KUKA KRL program: sPlanen2.src, sPlanen2.dat

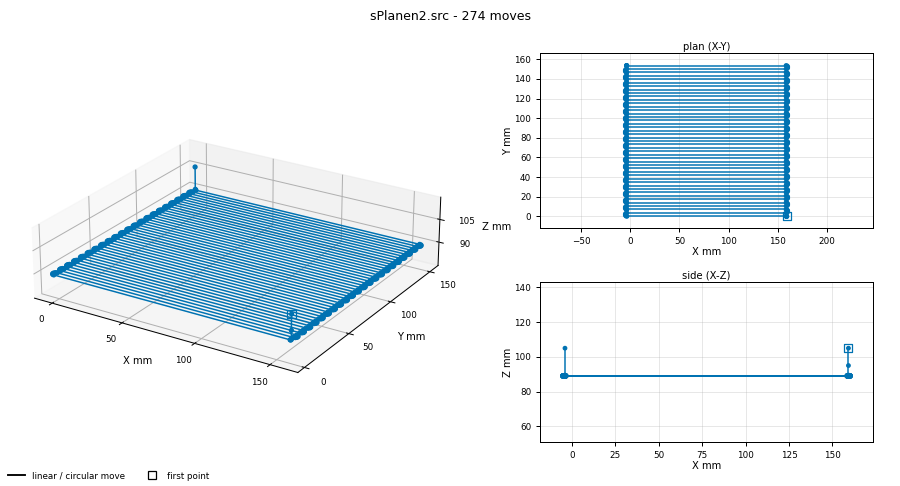
[picture p0: tool path of sPlanen2.src, 274 of 275 moves have a stored position in this frame; points joined in program order, loops and branches not executed]
--- sPlanen2.src ---
&ACCESS RVO
DEF sPlanen2()
; Generated by AUTODESK Fusion 360 CAM 2.0.14793
; Creation date: Thursday, March 16, 2023 18:51:23
;FOLD sPlanen2
; Start position (joint) = {A1 5,A2 -80,A3 100,A4 75,A5 -60,A6 -65}
; Tool Number            = 4
; Base Number            = 1
; Spindle Speed          = 5000 RPM
; Program file name      = sPlanen2.src

PTP {A1 5,A2 -80,A3 100,A4 75,A5 -60,A6 -65,E1 0,E2 0,E3 0,E4 0,E5 0,E6 0}
$VEL.CP=0.02
LIN {X 159.250,Y 0.025,Z 105.000,A 180.000,B 0.000,C 180.000} C_DIS
LIN {X 159.250,Y 0.025,Z 95.000,A 180.000,B 0.000,C 180.000} C_DIS
; Plunge Move Starts
$VEL.CP=0.01
LIN {X 159.250,Y 0.025,Z 89.500,A 180.000,B 0.000,C 180.000} C_DIS
; Lead In Move Starts
LIN {X 159.104,Y 0.025,Z 89.146,A 180.000,B 0.000,C 180.000} C_DIS
LIN {X 158.750,Y 0.025,Z 89.000,A 180.000,B 0.000,C 180.000} C_DIS
LIN {X 158.510,Y 0.025,Z 89.000,A 180.000,B 0.000,C 180.000} C_DIS
; Cutting Move Starts
$VEL.CP=0.02
LIN {X -3.510,Y 0.025,Z 89.000,A 180.000,B 0.000,C 180.000} C_DIS
; Link Move Starts
LIN {X -4.536,Y 0.358,Z 89.000,A 180.000,B 0.000,C 180.000} C_DIS
LIN {X -5.170,Y 1.231,Z 89.000,A 180.000,B 0.000,C 180.000} C_DIS
LIN {X -5.170,Y 2.309,Z 89.000,A 180.000,B 0.000,C 180.000} C_DIS
LIN {X -4.536,Y 3.182,Z 89.000,A 180.000,B 0.000,C 180.000} C_DIS
LIN {X -3.510,Y 3.515,Z 89.000,A 180.000,B 0.000,C 180.000} C_DIS
; Cutting Move Starts
LIN {X 158.510,Y 3.515,Z 89.000,A 180.000,B 0.000,C 180.000} C_DIS
; Link Move Starts
LIN {X 159.536,Y 3.848,Z 89.000,A 180.000,B 0.000,C 180.000} C_DIS
LIN {X 160.170,Y 4.721,Z 89.000,A 180.000,B 0.000,C 180.000} C_DIS
LIN {X 160.170,Y 5.800,Z 89.000,A 180.000,B 0.000,C 180.000} C_DIS
LIN {X 159.536,Y 6.672,Z 89.000,A 180.000,B 0.000,C 180.000} C_DIS
LIN {X 158.510,Y 7.005,Z 89.000,A 180.000,B 0.000,C 180.000} C_DIS
; Cutting Move Starts
LIN {X -3.510,Y 7.005,Z 89.000,A 180.000,B 0.000,C 180.000} C_DIS
; Link Move Starts
LIN {X -4.536,Y 7.339,Z 89.000,A 180.000,B 0.000,C 180.000} C_DIS
LIN {X -5.170,Y 8.211,Z 89.000,A 180.000,B 0.000,C 180.000} C_DIS
LIN {X -5.170,Y 9.290,Z 89.000,A 180.000,B 0.000,C 180.000} C_DIS
LIN {X -4.536,Y 10.162,Z 89.000,A 180.000,B 0.000,C 180.000} C_DIS
LIN {X -3.510,Y 10.495,Z 89.000,A 180.000,B 0.000,C 180.000} C_DIS
; Cutting Move Starts
LIN {X 158.510,Y 10.495,Z 89.000,A 180.000,B 0.000,C 180.000} C_DIS
; Link Move Starts
LIN {X 159.536,Y 10.829,Z 89.000,A 180.000,B 0.000,C 180.000} C_DIS
LIN {X 160.170,Y 11.701,Z 89.000,A 180.000,B 0.000,C 180.000} C_DIS
LIN {X 160.170,Y 12.780,Z 89.000,A 180.000,B 0.000,C 180.000} C_DIS
LIN {X 159.536,Y 13.652,Z 89.000,A 180.000,B 0.000,C 180.000} C_DIS
LIN {X 158.510,Y 13.986,Z 89.000,A 180.000,B 0.000,C 180.000} C_DIS
; Cutting Move Starts
LIN {X -3.510,Y 13.986,Z 89.000,A 180.000,B 0.000,C 180.000} C_DIS
; Link Move Starts
LIN {X -4.536,Y 14.319,Z 89.000,A 180.000,B 0.000,C 180.000} C_DIS
LIN {X -5.170,Y 15.191,Z 89.000,A 180.000,B 0.000,C 180.000} C_DIS
LIN {X -5.170,Y 16.270,Z 89.000,A 180.000,B 0.000,C 180.000} C_DIS
LIN {X -4.536,Y 17.142,Z 89.000,A 180.000,B 0.000,C 180.000} C_DIS
LIN {X -3.510,Y 17.476,Z 89.000,A 180.000,B 0.000,C 180.000} C_DIS
; Cutting Move Starts
LIN {X 158.510,Y 17.476,Z 89.000,A 180.000,B 0.000,C 180.000} C_DIS
; Link Move Starts
LIN {X 159.536,Y 17.809,Z 89.000,A 180.000,B 0.000,C 180.000} C_DIS
LIN {X 160.170,Y 18.681,Z 89.000,A 180.000,B 0.000,C 180.000} C_DIS
LIN {X 160.170,Y 19.760,Z 89.000,A 180.000,B 0.000,C 180.000} C_DIS
LIN {X 159.536,Y 20.633,Z 89.000,A 180.000,B 0.000,C 180.000} C_DIS
LIN {X 158.510,Y 20.966,Z 89.000,A 180.000,B 0.000,C 180.000} C_DIS
; Cutting Move Starts
LIN {X -3.510,Y 20.966,Z 89.000,A 180.000,B 0.000,C 180.000} C_DIS
; Link Move Starts
LIN {X -4.536,Y 21.299,Z 89.000,A 180.000,B 0.000,C 180.000} C_DIS
LIN {X -5.170,Y 22.172,Z 89.000,A 180.000,B 0.000,C 180.000} C_DIS
LIN {X -5.170,Y 23.250,Z 89.000,A 180.000,B 0.000,C 180.000} C_DIS
LIN {X -4.536,Y 24.123,Z 89.000,A 180.000,B 0.000,C 180.000} C_DIS
LIN {X -3.510,Y 24.456,Z 89.000,A 180.000,B 0.000,C 180.000} C_DIS
; Cutting Move Starts
LIN {X 158.510,Y 24.456,Z 89.000,A 180.000,B 0.000,C 180.000} C_DIS
; Link Move Starts
LIN {X 159.536,Y 24.789,Z 89.000,A 180.000,B 0.000,C 180.000} C_DIS
LIN {X 160.170,Y 25.662,Z 89.000,A 180.000,B 0.000,C 180.000} C_DIS
LIN {X 160.170,Y 26.740,Z 89.000,A 180.000,B 0.000,C 180.000} C_DIS
LIN {X 159.536,Y 27.613,Z 89.000,A 180.000,B 0.000,C 180.000} C_DIS
LIN {X 158.510,Y 27.946,Z 89.000,A 180.000,B 0.000,C 180.000} C_DIS
; Cutting Move Starts
LIN {X -3.510,Y 27.946,Z 89.000,A 180.000,B 0.000,C 180.000} C_DIS
; Link Move Starts
LIN {X -4.536,Y 28.279,Z 89.000,A 180.000,B 0.000,C 180.000} C_DIS
LIN {X -5.170,Y 29.152,Z 89.000,A 180.000,B 0.000,C 180.000} C_DIS
LIN {X -5.170,Y 30.230,Z 89.000,A 180.000,B 0.000,C 180.000} C_DIS
LIN {X -4.536,Y 31.103,Z 89.000,A 180.000,B 0.000,C 180.000} C_DIS
LIN {X -3.510,Y 31.436,Z 89.000,A 180.000,B 0.000,C 180.000} C_DIS
; Cutting Move Starts
LIN {X 158.510,Y 31.436,Z 89.000,A 180.000,B 0.000,C 180.000} C_DIS
; Link Move Starts
LIN {X 159.536,Y 31.769,Z 89.000,A 180.000,B 0.000,C 180.000} C_DIS
LIN {X 160.170,Y 32.642,Z 89.000,A 180.000,B 0.000,C 180.000} C_DIS
LIN {X 160.170,Y 33.720,Z 89.000,A 180.000,B 0.000,C 180.000} C_DIS
LIN {X 159.536,Y 34.593,Z 89.000,A 180.000,B 0.000,C 180.000} C_DIS
LIN {X 158.510,Y 34.926,Z 89.000,A 180.000,B 0.000,C 180.000} C_DIS
; Cutting Move Starts
LIN {X -3.510,Y 34.926,Z 89.000,A 180.000,B 0.000,C 180.000} C_DIS
; Link Move Starts
LIN {X -4.536,Y 35.259,Z 89.000,A 180.000,B 0.000,C 180.000} C_DIS
LIN {X -5.170,Y 36.132,Z 89.000,A 180.000,B 0.000,C 180.000} C_DIS
LIN {X -5.170,Y 37.211,Z 89.000,A 180.000,B 0.000,C 180.000} C_DIS
LIN {X -4.536,Y 38.083,Z 89.000,A 180.000,B 0.000,C 180.000} C_DIS
LIN {X -3.510,Y 38.416,Z 89.000,A 180.000,B 0.000,C 180.000} C_DIS
; Cutting Move Starts
LIN {X 158.510,Y 38.416,Z 89.000,A 180.000,B 0.000,C 180.000} C_DIS
; Link Move Starts
LIN {X 159.536,Y 38.750,Z 89.000,A 180.000,B 0.000,C 180.000} C_DIS
LIN {X 160.170,Y 39.622,Z 89.000,A 180.000,B 0.000,C 180.000} C_DIS
LIN {X 160.170,Y 40.701,Z 89.000,A 180.000,B 0.000,C 180.000} C_DIS
LIN {X 159.536,Y 41.573,Z 89.000,A 180.000,B 0.000,C 180.000} C_DIS
LIN {X 158.510,Y 41.906,Z 89.000,A 180.000,B 0.000,C 180.000} C_DIS
; Cutting Move Starts
LIN {X -3.510,Y 41.906,Z 89.000,A 180.000,B 0.000,C 180.000} C_DIS
; Link Move Starts
LIN {X -4.536,Y 42.240,Z 89.000,A 180.000,B 0.000,C 180.000} C_DIS
LIN {X -5.170,Y 43.112,Z 89.000,A 180.000,B 0.000,C 180.000} C_DIS
LIN {X -5.170,Y 44.191,Z 89.000,A 180.000,B 0.000,C 180.000} C_DIS
LIN {X -4.536,Y 45.063,Z 89.000,A 180.000,B 0.000,C 180.000} C_DIS
LIN {X -3.510,Y 45.397,Z 89.000,A 180.000,B 0.000,C 180.000} C_DIS
; Cutting Move Starts
LIN {X 158.510,Y 45.397,Z 89.000,A 180.000,B 0.000,C 180.000} C_DIS
; Link Move Starts
LIN {X 159.536,Y 45.730,Z 89.000,A 180.000,B 0.000,C 180.000} C_DIS
LIN {X 160.170,Y 46.602,Z 89.000,A 180.000,B 0.000,C 180.000} C_DIS
LIN {X 160.170,Y 47.681,Z 89.000,A 180.000,B 0.000,C 180.000} C_DIS
LIN {X 159.536,Y 48.553,Z 89.000,A 180.000,B 0.000,C 180.000} C_DIS
LIN {X 158.510,Y 48.887,Z 89.000,A 180.000,B 0.000,C 180.000} C_DIS
; Cutting Move Starts
LIN {X -3.510,Y 48.887,Z 89.000,A 180.000,B 0.000,C 180.000} C_DIS
; Link Move Starts
LIN {X -4.536,Y 49.220,Z 89.000,A 180.000,B 0.000,C 180.000} C_DIS
LIN {X -5.170,Y 50.092,Z 89.000,A 180.000,B 0.000,C 180.000} C_DIS
LIN {X -5.170,Y 51.171,Z 89.000,A 180.000,B 0.000,C 180.000} C_DIS
LIN {X -4.536,Y 52.044,Z 89.000,A 180.000,B 0.000,C 180.000} C_DIS
LIN {X -3.510,Y 52.377,Z 89.000,A 180.000,B 0.000,C 180.000} C_DIS
; Cutting Move Starts
LIN {X 158.510,Y 52.377,Z 89.000,A 180.000,B 0.000,C 180.000} C_DIS
; Link Move Starts
LIN {X 159.536,Y 52.710,Z 89.000,A 180.000,B 0.000,C 180.000} C_DIS
LIN {X 160.170,Y 53.583,Z 89.000,A 180.000,B 0.000,C 180.000} C_DIS
LIN {X 160.170,Y 54.661,Z 89.000,A 180.000,B 0.000,C 180.000} C_DIS
LIN {X 159.536,Y 55.534,Z 89.000,A 180.000,B 0.000,C 180.000} C_DIS
LIN {X 158.510,Y 55.867,Z 89.000,A 180.000,B 0.000,C 180.000} C_DIS
; Cutting Move Starts
LIN {X -3.510,Y 55.867,Z 89.000,A 180.000,B 0.000,C 180.000} C_DIS
; Link Move Starts
LIN {X -4.536,Y 56.200,Z 89.000,A 180.000,B 0.000,C 180.000} C_DIS
LIN {X -5.170,Y 57.073,Z 89.000,A 180.000,B 0.000,C 180.000} C_DIS
LIN {X -5.170,Y 58.151,Z 89.000,A 180.000,B 0.000,C 180.000} C_DIS
LIN {X -4.536,Y 59.024,Z 89.000,A 180.000,B 0.000,C 180.000} C_DIS
LIN {X -3.510,Y 59.357,Z 89.000,A 180.000,B 0.000,C 180.000} C_DIS
; Cutting Move Starts
LIN {X 158.510,Y 59.357,Z 89.000,A 180.000,B 0.000,C 180.000} C_DIS
; Link Move Starts
LIN {X 159.536,Y 59.690,Z 89.000,A 180.000,B 0.000,C 180.000} C_DIS
LIN {X 160.170,Y 60.563,Z 89.000,A 180.000,B 0.000,C 180.000} C_DIS
LIN {X 160.170,Y 61.641,Z 89.000,A 180.000,B 0.000,C 180.000} C_DIS
LIN {X 159.536,Y 62.514,Z 89.000,A 180.000,B 0.000,C 180.000} C_DIS
LIN {X 158.510,Y 62.847,Z 89.000,A 180.000,B 0.000,C 180.000} C_DIS
; Cutting Move Starts
LIN {X -3.510,Y 62.847,Z 89.000,A 180.000,B 0.000,C 180.000} C_DIS
; Link Move Starts
LIN {X -4.536,Y 63.180,Z 89.000,A 180.000,B 0.000,C 180.000} C_DIS
LIN {X -5.170,Y 64.053,Z 89.000,A 180.000,B 0.000,C 180.000} C_DIS
LIN {X -5.170,Y 65.131,Z 89.000,A 180.000,B 0.000,C 180.000} C_DIS
LIN {X -4.536,Y 66.004,Z 89.000,A 180.000,B 0.000,C 180.000} C_DIS
LIN {X -3.510,Y 66.337,Z 89.000,A 180.000,B 0.000,C 180.000} C_DIS
; Cutting Move Starts
LIN {X 158.510,Y 66.337,Z 89.000,A 180.000,B 0.000,C 180.000} C_DIS
; Link Move Starts
LIN {X 159.536,Y 66.670,Z 89.000,A 180.000,B 0.000,C 180.000} C_DIS
LIN {X 160.170,Y 67.543,Z 89.000,A 180.000,B 0.000,C 180.000} C_DIS
LIN {X 160.170,Y 68.622,Z 89.000,A 180.000,B 0.000,C 180.000} C_DIS
LIN {X 159.536,Y 69.494,Z 89.000,A 180.000,B 0.000,C 180.000} C_DIS
LIN {X 158.510,Y 69.827,Z 89.000,A 180.000,B 0.000,C 180.000} C_DIS
; Cutting Move Starts
LIN {X -3.510,Y 69.827,Z 89.000,A 180.000,B 0.000,C 180.000} C_DIS
; Link Move Starts
LIN {X -4.536,Y 70.161,Z 89.000,A 180.000,B 0.000,C 180.000} C_DIS
LIN {X -5.170,Y 71.033,Z 89.000,A 180.000,B 0.000,C 180.000} C_DIS
LIN {X -5.170,Y 72.112,Z 89.000,A 180.000,B 0.000,C 180.000} C_DIS
LIN {X -4.536,Y 72.984,Z 89.000,A 180.000,B 0.000,C 180.000} C_DIS
LIN {X -3.510,Y 73.317,Z 89.000,A 180.000,B 0.000,C 180.000} C_DIS
; Cutting Move Starts
LIN {X 158.510,Y 73.317,Z 89.000,A 180.000,B 0.000,C 180.000} C_DIS
; Link Move Starts
LIN {X 159.536,Y 73.651,Z 89.000,A 180.000,B 0.000,C 180.000} C_DIS
LIN {X 160.170,Y 74.523,Z 89.000,A 180.000,B 0.000,C 180.000} C_DIS
LIN {X 160.170,Y 75.602,Z 89.000,A 180.000,B 0.000,C 180.000} C_DIS
LIN {X 159.536,Y 76.474,Z 89.000,A 180.000,B 0.000,C 180.000} C_DIS
LIN {X 158.510,Y 76.808,Z 89.000,A 180.000,B 0.000,C 180.000} C_DIS
; Cutting Move Starts
LIN {X -3.510,Y 76.808,Z 89.000,A 180.000,B 0.000,C 180.000} C_DIS
; Link Move Starts
LIN {X -4.536,Y 77.141,Z 89.000,A 180.000,B 0.000,C 180.000} C_DIS
LIN {X -5.170,Y 78.013,Z 89.000,A 180.000,B 0.000,C 180.000} C_DIS
LIN {X -5.170,Y 79.092,Z 89.000,A 180.000,B 0.000,C 180.000} C_DIS
LIN {X -4.536,Y 79.964,Z 89.000,A 180.000,B 0.000,C 180.000} C_DIS
LIN {X -3.510,Y 80.298,Z 89.000,A 180.000,B 0.000,C 180.000} C_DIS
; Cutting Move Starts
LIN {X 158.510,Y 80.298,Z 89.000,A 180.000,B 0.000,C 180.000} C_DIS
; Link Move Starts
LIN {X 159.536,Y 80.631,Z 89.000,A 180.000,B 0.000,C 180.000} C_DIS
LIN {X 160.170,Y 81.503,Z 89.000,A 180.000,B 0.000,C 180.000} C_DIS
LIN {X 160.170,Y 82.582,Z 89.000,A 180.000,B 0.000,C 180.000} C_DIS
LIN {X 159.536,Y 83.455,Z 89.000,A 180.000,B 0.000,C 180.000} C_DIS
LIN {X 158.510,Y 83.788,Z 89.000,A 180.000,B 0.000,C 180.000} C_DIS
; Cutting Move Starts
LIN {X -3.510,Y 83.788,Z 89.000,A 180.000,B 0.000,C 180.000} C_DIS
; Link Move Starts
LIN {X -4.536,Y 84.121,Z 89.000,A 180.000,B 0.000,C 180.000} C_DIS
LIN {X -5.170,Y 84.994,Z 89.000,A 180.000,B 0.000,C 180.000} C_DIS
LIN {X -5.170,Y 86.072,Z 89.000,A 180.000,B 0.000,C 180.000} C_DIS
LIN {X -4.536,Y 86.945,Z 89.000,A 180.000,B 0.000,C 180.000} C_DIS
LIN {X -3.510,Y 87.278,Z 89.000,A 180.000,B 0.000,C 180.000} C_DIS
; Cutting Move Starts
LIN {X 158.510,Y 87.278,Z 89.000,A 180.000,B 0.000,C 180.000} C_DIS
; Link Move Starts
LIN {X 159.536,Y 87.611,Z 89.000,A 180.000,B 0.000,C 180.000} C_DIS
LIN {X 160.170,Y 88.484,Z 89.000,A 180.000,B 0.000,C 180.000} C_DIS
LIN {X 160.170,Y 89.562,Z 89.000,A 180.000,B 0.000,C 180.000} C_DIS
LIN {X 159.536,Y 90.435,Z 89.000,A 180.000,B 0.000,C 180.000} C_DIS
LIN {X 158.510,Y 90.768,Z 89.000,A 180.000,B 0.000,C 180.000} C_DIS
; Cutting Move Starts
LIN {X -3.510,Y 90.768,Z 89.000,A 180.000,B 0.000,C 180.000} C_DIS
; Link Move Starts
LIN {X -4.536,Y 91.101,Z 89.000,A 180.000,B 0.000,C 180.000} C_DIS
LIN {X -5.170,Y 91.974,Z 89.000,A 180.000,B 0.000,C 180.000} C_DIS
LIN {X -5.170,Y 93.052,Z 89.000,A 180.000,B 0.000,C 180.000} C_DIS
LIN {X -4.536,Y 93.925,Z 89.000,A 180.000,B 0.000,C 180.000} C_DIS
LIN {X -3.510,Y 94.258,Z 89.000,A 180.000,B 0.000,C 180.000} C_DIS
; Cutting Move Starts
LIN {X 158.510,Y 94.258,Z 89.000,A 180.000,B 0.000,C 180.000} C_DIS
; Link Move Starts
LIN {X 159.536,Y 94.591,Z 89.000,A 180.000,B 0.000,C 180.000} C_DIS
LIN {X 160.170,Y 95.464,Z 89.000,A 180.000,B 0.000,C 180.000} C_DIS
LIN {X 160.170,Y 96.542,Z 89.000,A 180.000,B 0.000,C 180.000} C_DIS
LIN {X 159.536,Y 97.415,Z 89.000,A 180.000,B 0.000,C 180.000} C_DIS
LIN {X 158.510,Y 97.748,Z 89.000,A 180.000,B 0.000,C 180.000} C_DIS
; Cutting Move Starts
LIN {X -3.510,Y 97.748,Z 89.000,A 180.000,B 0.000,C 180.000} C_DIS
; Link Move Starts
LIN {X -4.536,Y 98.081,Z 89.000,A 180.000,B 0.000,C 180.000} C_DIS
LIN {X -5.170,Y 98.954,Z 89.000,A 180.000,B 0.000,C 180.000} C_DIS
LIN {X -5.170,Y 100.033,Z 89.000,A 180.000,B 0.000,C 180.000} C_DIS
LIN {X -4.536,Y 100.905,Z 89.000,A 180.000,B 0.000,C 180.000} C_DIS
LIN {X -3.510,Y 101.238,Z 89.000,A 180.000,B 0.000,C 180.000} C_DIS
; Cutting Move Starts
LIN {X 158.510,Y 101.238,Z 89.000,A 180.000,B 0.000,C 180.000} C_DIS
; Link Move Starts
LIN {X 159.536,Y 101.572,Z 89.000,A 180.000,B 0.000,C 180.000} C_DIS
LIN {X 160.170,Y 102.444,Z 89.000,A 180.000,B 0.000,C 180.000} C_DIS
LIN {X 160.170,Y 103.523,Z 89.000,A 180.000,B 0.000,C 180.000} C_DIS
LIN {X 159.536,Y 104.395,Z 89.000,A 180.000,B 0.000,C 180.000} C_DIS
LIN {X 158.510,Y 104.728,Z 89.000,A 180.000,B 0.000,C 180.000} C_DIS
; Cutting Move Starts
LIN {X -3.510,Y 104.728,Z 89.000,A 180.000,B 0.000,C 180.000} C_DIS
; Link Move Starts
LIN {X -4.536,Y 105.062,Z 89.000,A 180.000,B 0.000,C 180.000} C_DIS
LIN {X -5.170,Y 105.934,Z 89.000,A 180.000,B 0.000,C 180.000} C_DIS
LIN {X -5.170,Y 107.013,Z 89.000,A 180.000,B 0.000,C 180.000} C_DIS
LIN {X -4.536,Y 107.885,Z 89.000,A 180.000,B 0.000,C 180.000} C_DIS
LIN {X -3.510,Y 108.219,Z 89.000,A 180.000,B 0.000,C 180.000} C_DIS
; Cutting Move Starts
LIN {X 158.510,Y 108.219,Z 89.000,A 180.000,B 0.000,C 180.000} C_DIS
; Link Move Starts
LIN {X 159.536,Y 108.552,Z 89.000,A 180.000,B 0.000,C 180.000} C_DIS
LIN {X 160.170,Y 109.424,Z 89.000,A 180.000,B 0.000,C 180.000} C_DIS
LIN {X 160.170,Y 110.503,Z 89.000,A 180.000,B 0.000,C 180.000} C_DIS
LIN {X 159.536,Y 111.375,Z 89.000,A 180.000,B 0.000,C 180.000} C_DIS
LIN {X 158.510,Y 111.709,Z 89.000,A 180.000,B 0.000,C 180.000} C_DIS
; Cutting Move Starts
LIN {X -3.510,Y 111.709,Z 89.000,A 180.000,B 0.000,C 180.000} C_DIS
; Link Move Starts
LIN {X -4.536,Y 112.042,Z 89.000,A 180.000,B 0.000,C 180.000} C_DIS
LIN {X -5.170,Y 112.914,Z 89.000,A 180.000,B 0.000,C 180.000} C_DIS
LIN {X -5.170,Y 113.993,Z 89.000,A 180.000,B 0.000,C 180.000} C_DIS
LIN {X -4.536,Y 114.866,Z 89.000,A 180.000,B 0.000,C 180.000} C_DIS
LIN {X -3.510,Y 115.199,Z 89.000,A 180.000,B 0.000,C 180.000} C_DIS
; Cutting Move Starts
LIN {X 158.510,Y 115.199,Z 89.000,A 180.000,B 0.000,C 180.000} C_DIS
; Link Move Starts
LIN {X 159.536,Y 115.532,Z 89.000,A 180.000,B 0.000,C 180.000} C_DIS
LIN {X 160.170,Y 116.405,Z 89.000,A 180.000,B 0.000,C 180.000} C_DIS
LIN {X 160.170,Y 117.483,Z 89.000,A 180.000,B 0.000,C 180.000} C_DIS
LIN {X 159.536,Y 118.356,Z 89.000,A 180.000,B 0.000,C 180.000} C_DIS
LIN {X 158.510,Y 118.689,Z 89.000,A 180.000,B 0.000,C 180.000} C_DIS
; Cutting Move Starts
LIN {X -3.510,Y 118.689,Z 89.000,A 180.000,B 0.000,C 180.000} C_DIS
; Link Move Starts
LIN {X -4.536,Y 119.022,Z 89.000,A 180.000,B 0.000,C 180.000} C_DIS
LIN {X -5.170,Y 119.895,Z 89.000,A 180.000,B 0.000,C 180.000} C_DIS
LIN {X -5.170,Y 120.973,Z 89.000,A 180.000,B 0.000,C 180.000} C_DIS
LIN {X -4.536,Y 121.846,Z 89.000,A 180.000,B 0.000,C 180.000} C_DIS
LIN {X -3.510,Y 122.179,Z 89.000,A 180.000,B 0.000,C 180.000} C_DIS
; Cutting Move Starts
LIN {X 158.510,Y 122.179,Z 89.000,A 180.000,B 0.000,C 180.000} C_DIS
; Link Move Starts
LIN {X 159.536,Y 122.512,Z 89.000,A 180.000,B 0.000,C 180.000} C_DIS
LIN {X 160.170,Y 123.385,Z 89.000,A 180.000,B 0.000,C 180.000} C_DIS
LIN {X 160.170,Y 124.463,Z 89.000,A 180.000,B 0.000,C 180.000} C_DIS
LIN {X 159.536,Y 125.336,Z 89.000,A 180.000,B 0.000,C 180.000} C_DIS
LIN {X 158.510,Y 125.669,Z 89.000,A 180.000,B 0.000,C 180.000} C_DIS
; Cutting Move Starts
LIN {X -3.510,Y 125.669,Z 89.000,A 180.000,B 0.000,C 180.000} C_DIS
; Link Move Starts
LIN {X -4.536,Y 126.002,Z 89.000,A 180.000,B 0.000,C 180.000} C_DIS
LIN {X -5.170,Y 126.875,Z 89.000,A 180.000,B 0.000,C 180.000} C_DIS
LIN {X -5.170,Y 127.953,Z 89.000,A 180.000,B 0.000,C 180.000} C_DIS
LIN {X -4.536,Y 128.826,Z 89.000,A 180.000,B 0.000,C 180.000} C_DIS
LIN {X -3.510,Y 129.159,Z 89.000,A 180.000,B 0.000,C 180.000} C_DIS
; Cutting Move Starts
LIN {X 158.510,Y 129.159,Z 89.000,A 180.000,B 0.000,C 180.000} C_DIS
; Link Move Starts
LIN {X 159.536,Y 129.493,Z 89.000,A 180.000,B 0.000,C 180.000} C_DIS
LIN {X 160.170,Y 130.365,Z 89.000,A 180.000,B 0.000,C 180.000} C_DIS
LIN {X 160.170,Y 131.444,Z 89.000,A 180.000,B 0.000,C 180.000} C_DIS
LIN {X 159.536,Y 132.316,Z 89.000,A 180.000,B 0.000,C 180.000} C_DIS
LIN {X 158.510,Y 132.649,Z 89.000,A 180.000,B 0.000,C 180.000} C_DIS
; Cutting Move Starts
LIN {X -3.510,Y 132.649,Z 89.000,A 180.000,B 0.000,C 180.000} C_DIS
; Link Move Starts
LIN {X -4.536,Y 132.983,Z 89.000,A 180.000,B 0.000,C 180.000} C_DIS
LIN {X -5.170,Y 133.855,Z 89.000,A 180.000,B 0.000,C 180.000} C_DIS
LIN {X -5.170,Y 134.934,Z 89.000,A 180.000,B 0.000,C 180.000} C_DIS
LIN {X -4.536,Y 135.806,Z 89.000,A 180.000,B 0.000,C 180.000} C_DIS
LIN {X -3.510,Y 136.139,Z 89.000,A 180.000,B 0.000,C 180.000} C_DIS
; Cutting Move Starts
LIN {X 158.510,Y 136.139,Z 89.000,A 180.000,B 0.000,C 180.000} C_DIS
; Link Move Starts
LIN {X 159.536,Y 136.473,Z 89.000,A 180.000,B 0.000,C 180.000} C_DIS
LIN {X 160.170,Y 137.345,Z 89.000,A 180.000,B 0.000,C 180.000} C_DIS
LIN {X 160.170,Y 138.424,Z 89.000,A 180.000,B 0.000,C 180.000} C_DIS
LIN {X 159.536,Y 139.296,Z 89.000,A 180.000,B 0.000,C 180.000} C_DIS
LIN {X 158.510,Y 139.630,Z 89.000,A 180.000,B 0.000,C 180.000} C_DIS
; Cutting Move Starts
LIN {X -3.510,Y 139.630,Z 89.000,A 180.000,B 0.000,C 180.000} C_DIS
; Link Move Starts
LIN {X -4.536,Y 139.963,Z 89.000,A 180.000,B 0.000,C 180.000} C_DIS
LIN {X -5.170,Y 140.835,Z 89.000,A 180.000,B 0.000,C 180.000} C_DIS
LIN {X -5.170,Y 141.914,Z 89.000,A 180.000,B 0.000,C 180.000} C_DIS
LIN {X -4.536,Y 142.786,Z 89.000,A 180.000,B 0.000,C 180.000} C_DIS
LIN {X -3.510,Y 143.120,Z 89.000,A 180.000,B 0.000,C 180.000} C_DIS
; Cutting Move Starts
LIN {X 158.510,Y 143.120,Z 89.000,A 180.000,B 0.000,C 180.000} C_DIS
; Link Move Starts
LIN {X 159.536,Y 143.453,Z 89.000,A 180.000,B 0.000,C 180.000} C_DIS
LIN {X 160.170,Y 144.325,Z 89.000,A 180.000,B 0.000,C 180.000} C_DIS
LIN {X 160.170,Y 145.404,Z 89.000,A 180.000,B 0.000,C 180.000} C_DIS
LIN {X 159.536,Y 146.276,Z 89.000,A 180.000,B 0.000,C 180.000} C_DIS
LIN {X 158.510,Y 146.610,Z 89.000,A 180.000,B 0.000,C 180.000} C_DIS
; Cutting Move Starts
LIN {X -3.510,Y 146.610,Z 89.000,A 180.000,B 0.000,C 180.000} C_DIS
; Link Move Starts
LIN {X -4.536,Y 146.943,Z 89.000,A 180.000,B 0.000,C 180.000} C_DIS
LIN {X -5.170,Y 147.816,Z 89.000,A 180.000,B 0.000,C 180.000} C_DIS
LIN {X -5.170,Y 148.894,Z 89.000,A 180.000,B 0.000,C 180.000} C_DIS
LIN {X -4.536,Y 149.767,Z 89.000,A 180.000,B 0.000,C 180.000} C_DIS
LIN {X -3.510,Y 150.100,Z 89.000,A 180.000,B 0.000,C 180.000} C_DIS
; Cutting Move Starts
LIN {X 158.510,Y 150.100,Z 89.000,A 180.000,B 0.000,C 180.000} C_DIS
; Link Move Starts
LIN {X 159.536,Y 150.433,Z 89.000,A 180.000,B 0.000,C 180.000} C_DIS
LIN {X 160.170,Y 151.306,Z 89.000,A 180.000,B 0.000,C 180.000} C_DIS
LIN {X 160.170,Y 152.384,Z 89.000,A 180.000,B 0.000,C 180.000} C_DIS
LIN {X 159.536,Y 153.257,Z 89.000,A 180.000,B 0.000,C 180.000} C_DIS
LIN {X 158.510,Y 153.590,Z 89.000,A 180.000,B 0.000,C 180.000} C_DIS
; Cutting Move Starts
LIN {X -3.510,Y 153.590,Z 89.000,A 180.000,B 0.000,C 180.000} C_DIS
; Lead Out Move Starts
LIN {X -3.864,Y 153.590,Z 89.146,A 180.000,B 0.000,C 180.000} C_DIS
LIN {X -4.010,Y 153.590,Z 89.500,A 180.000,B 0.000,C 180.000} C_DIS
; Rapid Move Starts
LIN {X -4.010,Y 153.590,Z 105.000,A 180.000,B 0.000,C 180.000} C_DIS
;ENDFOLD
END

--- sPlanen2.dat ---
&ACCESS RVO
DEFDAT sPlanen2
;FOLD EXTERNAL DECLARATIONS;%{PE}%MKUKATPBASIS,%CEXT,%VCOMMON,%P
  ;FOLD BASISTECH EXT;%{PE}%MKUKATPBASIS,%CEXT,%VEXT,%P
    EXT  BAS (BAS_COMMAND  :IN,REAL  :IN )
  ;ENDFOLD (BASISTECH EXT)

;ENDFOLD (EXTERNAL DECLARATIONS)
ENDDAT
